SUBAPPLICATION Sorter (* Subapplication Type *)
  (* Standard: 61499-2 *)
  (* Version 1.0, 2022-11-15, Maximilian Scharf *)
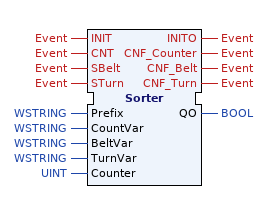
  EVENT_INPUT
    INIT;
    CNT;
    SBelt;
    STurn;
  END_EVENT
  EVENT_OUTPUT
    INITO;
    CNF_Counter;
    CNF_Belt;
    CNF_Turn;
  END_EVENT
  VAR_INPUT
    Prefix : WSTRING;
    CountVar : WSTRING;
    BeltVar : WSTRING;
    TurnVar : WSTRING;
    Counter : UINT;
  END_VAR
  VAR_OUTPUT
    QO : BOOL;
  END_VAR
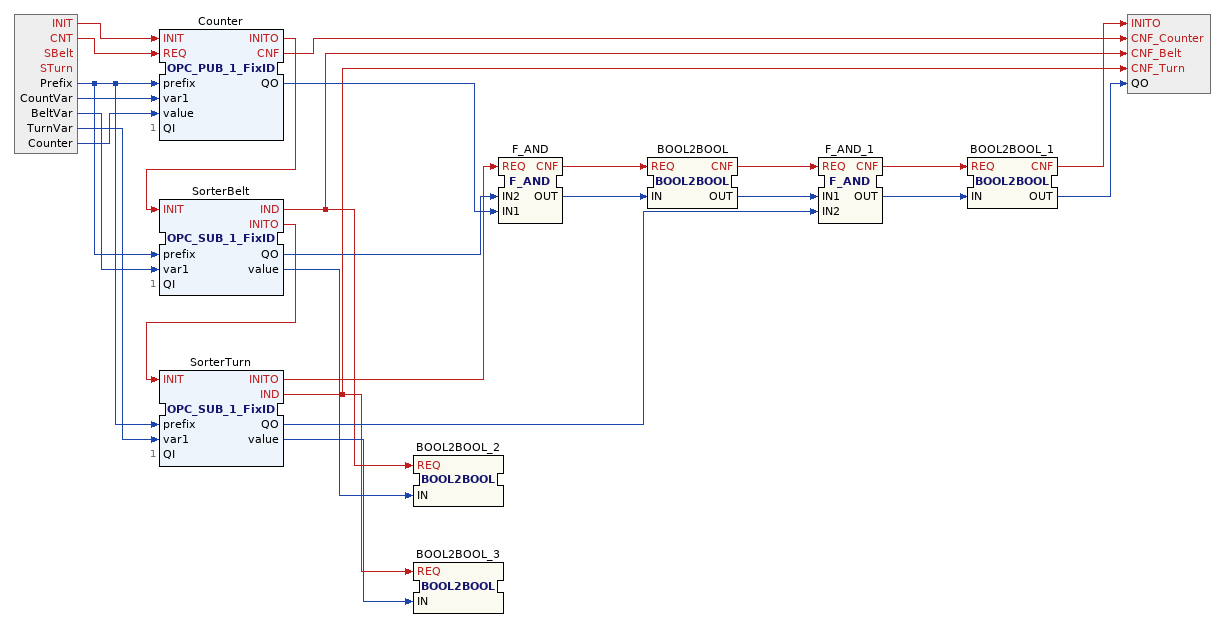
  FBS
    F_AND : F_AND;
    F_AND_1 : F_AND;
    BOOL2BOOL : BOOL2BOOL;
    BOOL2BOOL_1 : BOOL2BOOL;
    BOOL2BOOL_2 : BOOL2BOOL;
    BOOL2BOOL_3 : BOOL2BOOL;
  END_FBS
  SUBAPPS
    SorterBelt : OPC_SUB_1_FixID(QI := 1);
    SorterTurn : OPC_SUB_1_FixID(QI := 1);
    Counter : OPC_PUB_1_FixID(QI := 1);
  END_SUBAPPS
  EVENT_CONNECTIONS
    F_AND.CNF TO BOOL2BOOL.REQ;
    BOOL2BOOL.CNF TO F_AND_1.REQ;
    F_AND_1.CNF TO BOOL2BOOL_1.REQ;
    BOOL2BOOL_1.CNF TO INITO;
    SorterBelt.IND TO CNF_Belt;
    SorterBelt.INITO TO SorterTurn.INIT;
    SorterTurn.INITO TO F_AND.REQ;
    SorterTurn.IND TO CNF_Turn;
    SorterBelt.IND TO BOOL2BOOL_2.REQ;
    SorterTurn.IND TO BOOL2BOOL_3.REQ;
    INIT TO Counter.INIT;
    Counter.INITO TO SorterBelt.INIT;
    Counter.CNF TO CNF_Counter;
    CNT TO Counter.REQ;
  END_CONNECTIONS
  DATA_CONNECTIONS
    F_AND.OUT TO BOOL2BOOL.IN;
    BOOL2BOOL.OUT TO F_AND_1.IN1;
    F_AND_1.OUT TO BOOL2BOOL_1.IN;
    BOOL2BOOL_1.OUT TO QO;
    Prefix TO SorterBelt.prefix;
    BeltVar TO SorterBelt.var1;
    SorterBelt.QO TO F_AND.IN2;
    Prefix TO SorterTurn.prefix;
    TurnVar TO SorterTurn.var1;
    SorterTurn.QO TO F_AND_1.IN2;
    SorterBelt.value TO BOOL2BOOL_2.IN;
    SorterTurn.value TO BOOL2BOOL_3.IN;
    Prefix TO Counter.prefix;
    CountVar TO Counter.var1;
    Counter.QO TO F_AND.IN1;
    Counter TO Counter.value;
  END_CONNECTIONS
END_SUBAPPLICATION
